TYPE ST_IntToBool :
UNION
	nInt : INT:=1;
	BitList : ST_BoolList;
END_UNION
END_TYPE

(* stored: Version 1.1.0.1, ProductVersion 3.1.4024.13
   DUT ST_IntToBool: Id {55e752fc-67a7-475e-9c81-47554083f232} *)
